{attribute 'qualified_only'}
VAR_GLOBAL
END_VAR

(* stored: Version 1.1.0.1, ProductVersion 3.1.4024.15
   GVL GVL_Global: Id {97eb74c7-52db-4abf-af7b-07232158a512} *)
